PROGRAM P1_02_Batch
VAR
	fbBatch					:FB_Batch;
	fbBatchLog				:FB_BatchLog;
END_VAR
VAR // added by the converter: edge detectors and wires of the graphical bodies
    _rt1, _rt2, _rt3 : R_TRIG;
END_VAR

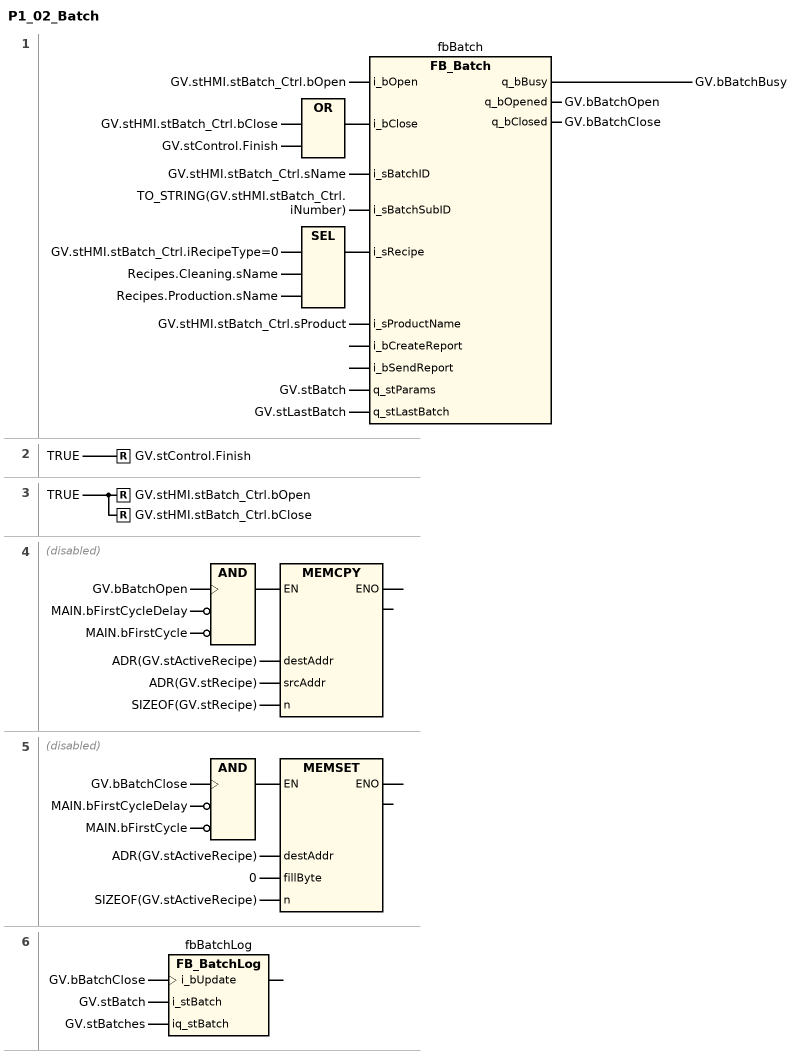
// NETWORK 1
fbBatch(
    i_bOpen := GV.stHMI.stBatch_Ctrl.bOpen,
    i_bClose := GV.stHMI.stBatch_Ctrl.bClose OR GV.stControl.Finish,
    i_sBatchID := GV.stHMI.stBatch_Ctrl.sName,
    i_sBatchSubID := TO_STRING(GV.stHMI.stBatch_Ctrl.iNumber),
    i_sRecipe := SEL(GV.stHMI.stBatch_Ctrl.iRecipeType=0, Recipes.Cleaning.sName, Recipes.Production.sName),
    i_sProductName := GV.stHMI.stBatch_Ctrl.sProduct,
    q_stParams := GV.stBatch,
    q_stLastBatch := GV.stLastBatch,
    q_bOpened => GV.bBatchOpen,
    q_bClosed => GV.bBatchClose); // FB_Batch
GV.bBatchBusy := fbBatch.q_bBusy;

// NETWORK 2
GV.stControl.Finish R= TRUE;

// NETWORK 3
GV.stHMI.stBatch_Ctrl.bOpen R= TRUE;
GV.stHMI.stBatch_Ctrl.bClose R= TRUE;

// NETWORK 4 (disabled)
// _rt1(CLK := GV.bBatchOpen);
// IF _rt1.Q AND NOT MAIN.bFirstCycleDelay AND NOT MAIN.bFirstCycle THEN
//     MEMCPY(destAddr := ADR(GV.stActiveRecipe), srcAddr := ADR(GV.stRecipe), n := SIZEOF(GV.stRecipe));
// END_IF

// NETWORK 5 (disabled)
// _rt2(CLK := GV.bBatchClose);
// IF _rt2.Q AND NOT MAIN.bFirstCycleDelay AND NOT MAIN.bFirstCycle THEN
//     MEMSET(destAddr := ADR(GV.stActiveRecipe), fillByte := 0, n := SIZEOF(GV.stActiveRecipe));
// END_IF

// NETWORK 6
_rt3(CLK := GV.bBatchClose);
fbBatchLog(i_bUpdate := _rt3.Q, i_stBatch := GV.stBatch, iq_stBatch := GV.stBatches); // FB_BatchLog

END_PROGRAM

(* stored: Version 1.1.0.1
   POU P1_02_Batch: Id {fde4e061-7102-4637-ad9f-2ce99741e8b7}, SpecialFunc None *)
